INTERFACE I_PullWheels EXTENDS I_Module, I_TaskResult, I_Resettable, I_Override, I_ContainStatemachine

PROPERTY PullWheelCylinder : I_Cylinder
GET
END_GET
END_PROPERTY

PROPERTY PullWheelLeftAxis : I_Mc2Axis_PTP
GET
END_GET
END_PROPERTY

PROPERTY PullWheelRightAxis : I_Mc2SlaveAxis
GET
END_GET
END_PROPERTY

PROPERTY Recipe : REFERENCE TO ST_PullWheelsRecipe
GET
END_GET
END_PROPERTY

END_INTERFACE

(* stored: Version 1.1.0.1, ProductVersion 3.1.4026.20
   Itf I_PullWheels: Id {c9baefc0-4f3f-4a56-bc84-a806f315d77b}
   Property PullWheelCylinder: Id {c32ebd20-10d4-4df8-89f9-7f9444c19250}
   Get Get: Id {237b2cc9-06b3-46b7-86c9-d69e0b289357}
   Property PullWheelLeftAxis: Id {e3c7b426-2737-40e2-992f-f86fc3f0cc6a}
   Get Get: Id {294fd62f-f942-49dc-9c33-59b971441ebd}
   Property PullWheelRightAxis: Id {46e7cce9-ba13-40ee-a7e9-ad3978f4489a}
   Get Get: Id {994c8324-d3a4-4433-950e-b3c118effcbf}
   Property Recipe: Id {3d5677f2-ca34-4269-a185-a1e1c919e7c8}
   Get Get: Id {822a6524-9eef-4a3a-b73c-cceda396c1c0} *)
